// TIA Portal V20 export
FUNCTION_BLOCK "FB_Digital_Output"   // FB3, LAD
{ S7_Optimized_Access := 'TRUE' }
// stored: AutoNumber false, MemoryReserve 100, SetENOAutomatically false
   VAR_INPUT
      DB_In_Emergency_Stop_Release : Bool;
      DB_In_Selected_Voltage_220V : Bool;
      DB_In_Selected_Voltage_127V : Bool;
      DB_Spin_Carousel_Frequency_Inverter_Speed_1 : Bool;
      DB_Spin_Carousel_Frequency_Inverter_Speed_2 : Bool;
      DB_Spin_Carousel_Frequency_Inverter_Speed_3 : Bool;
      DB_Conveyor_Belt_Frequency_Inverter_Speed_1 : Bool;
      DB_Conveyor_Belt_Frequency_Inverter_Speed_2 : Bool;
      DB_Conveyor_Belt_Frequency_Inverter_Speed_3 : Bool;
      DB_Turn_On_Conveyor_Belt_Motor_Spinner_Get_Entrace_Function_Test : Bool;
      DB_Turn_On_Conveyor_Belt_Motor_Rework_Conveyor_Belt_Get_Entrace_Functional_Test : Bool;
      DB_Turn_On_Conveyor_Belt_Motor_Spinner_Get_Exit_Functional_Test : Bool;
      DB_Turn_On_Conveyor_Belt_Motor_Rework_Conveyor_Belt_Get_Exit_Funcional_Test : Bool;
      DB_Open_Air_Pressure : Bool;
      DB_Valve_Advance_Spinner_Get_Entrace_Functional_Test : Bool;
      DB_Valve_Advance_Spinner_Get_Exit_Functional_Test : Bool;
      DB_Signal_Pre_Functional_Test_Production_Line : Bool;
      DB_Digital_Output_14 : Bool;
      DB_Digital_Output_15 : Bool;
      DB_Digital_Output_16 : Bool;
      DB_Digital_Output_17 : Bool;
      DB_Digital_Output_18 : Bool;
      DB_Digital_Output_19 : Bool;
      DB_Digital_Output_20 : Bool;
      DB_Digital_Output_21 : Bool;
      DB_Digital_Output_22 : Bool;
      DB_Digital_Output_23 : Bool;
      DB_Voltage_220V_Selected : Bool;
      DB_Voltage_127V_Selected : Bool;
   END_VAR
   VAR_OUTPUT
      DO_Spin_Carousel_Frequency_Inverter_Speed_1 : Bool;
      DO_Spin_Carousel_Frequency_Inverter_Speed_2 : Bool;
      DO_Spin_Carousel_Frequency_Inverter_Speed_3 : Bool;
      DO_Conveyor_Belt_Frequency_Inverter_Speed_1 : Bool;
      DO_Conveyor_Belt_Frequency_Inverter_Speed_2 : Bool;
      DO_Conveyor_Belt_Frequency_Inverter_Speed_3 : Bool;
      DO_Turn_On_Conveyor_Belt_Motor_Spinner_Get_Entrace_Function_Test : Bool;
      DO_Turn_On_Conveyor_Belt_Motor_Rework_Conveyor_Belt_Get_Entrace_Functional_Test : Bool;
      DO_Turn_On_Conveyor_Belt_Motor_Spinner_Get_Exit_Functional_Test : Bool;
      DO_Turn_On_Conveyor_Belt_Motor_Rework_Conveyor_Belt_Get_Exit_Funcional_Test : Bool;
      DO_Open_Air_Pressure : Bool;
      DO_Valve_Advance_Spinner_Entrace_Functional_Test : Bool;
      DO_Valve_Advance_Spinner_Exit_Functional_Test : Bool;
      DO_Signal_Pre_Functional_Test_Production_Line : Bool;
      DO_Digital_Output_14 : Bool;
      DO_Digital_Output_15 : Bool;
      DO_Digital_Output_16 : Bool;
      DO_Digital_Output_17 : Bool;
      DO_Digital_Output_18 : Bool;
      DO_Digital_Output_19 : Bool;
      DO_Digital_Output_20 : Bool;
      DO_Digital_Output_21 : Bool;
      DO_Digital_Output_22 : Bool;
      DO_Digital_Output_23 : Bool;
      DO_Voltage_220V_Selected : Bool;
      DO_Voltage_127V_Selected : Bool;
   END_VAR
   VAR
      Timer_Delay_Turn_On_220_V { S7_SetPoint := 'True'} : TON_TIME;
      Timer_Delay_Turn_On_127_V { S7_SetPoint := 'True'} : TON_TIME;
   END_VAR
BEGIN

REGION Network 1
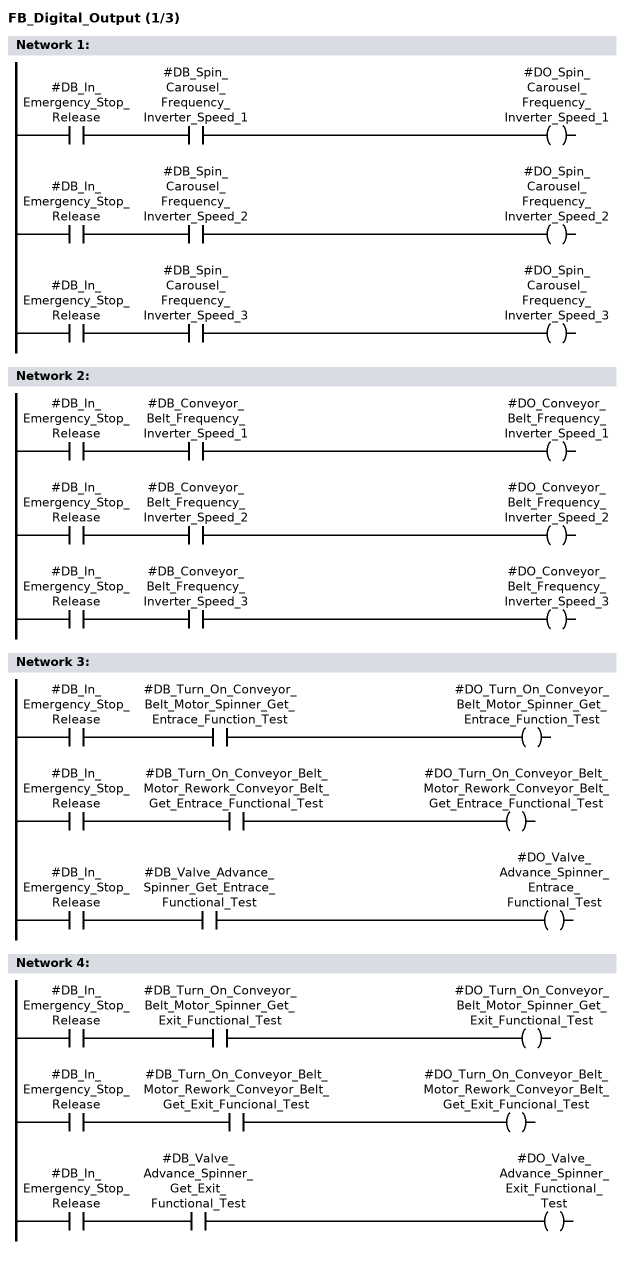
   RUNG wire#powerrail
      Contact( #DB_In_Emergency_Stop_Release )
      Contact( #DB_Spin_Carousel_Frequency_Inverter_Speed_1 )
      Coil( #DO_Spin_Carousel_Frequency_Inverter_Speed_1 )
   END_RUNG
   RUNG wire#powerrail
      Contact( #DB_In_Emergency_Stop_Release )
      Contact( #DB_Spin_Carousel_Frequency_Inverter_Speed_2 )
      Coil( #DO_Spin_Carousel_Frequency_Inverter_Speed_2 )
   END_RUNG
   RUNG wire#powerrail
      Contact( #DB_In_Emergency_Stop_Release )
      Contact( #DB_Spin_Carousel_Frequency_Inverter_Speed_3 )
      Coil( #DO_Spin_Carousel_Frequency_Inverter_Speed_3 )
   END_RUNG
   // the same network as SCL:
   #DO_Spin_Carousel_Frequency_Inverter_Speed_1 := #DB_In_Emergency_Stop_Release AND #DB_Spin_Carousel_Frequency_Inverter_Speed_1;
   #DO_Spin_Carousel_Frequency_Inverter_Speed_2 := #DB_In_Emergency_Stop_Release AND #DB_Spin_Carousel_Frequency_Inverter_Speed_2;
   #DO_Spin_Carousel_Frequency_Inverter_Speed_3 := #DB_In_Emergency_Stop_Release AND #DB_Spin_Carousel_Frequency_Inverter_Speed_3;
END_REGION

REGION Network 2
   RUNG wire#powerrail
      Contact( #DB_In_Emergency_Stop_Release )
      Contact( #DB_Conveyor_Belt_Frequency_Inverter_Speed_1 )
      Coil( #DO_Conveyor_Belt_Frequency_Inverter_Speed_1 )
   END_RUNG
   RUNG wire#powerrail
      Contact( #DB_In_Emergency_Stop_Release )
      Contact( #DB_Conveyor_Belt_Frequency_Inverter_Speed_2 )
      Coil( #DO_Conveyor_Belt_Frequency_Inverter_Speed_2 )
   END_RUNG
   RUNG wire#powerrail
      Contact( #DB_In_Emergency_Stop_Release )
      Contact( #DB_Conveyor_Belt_Frequency_Inverter_Speed_3 )
      Coil( #DO_Conveyor_Belt_Frequency_Inverter_Speed_3 )
   END_RUNG
   // the same network as SCL:
   #DO_Conveyor_Belt_Frequency_Inverter_Speed_1 := #DB_In_Emergency_Stop_Release AND #DB_Conveyor_Belt_Frequency_Inverter_Speed_1;
   #DO_Conveyor_Belt_Frequency_Inverter_Speed_2 := #DB_In_Emergency_Stop_Release AND #DB_Conveyor_Belt_Frequency_Inverter_Speed_2;
   #DO_Conveyor_Belt_Frequency_Inverter_Speed_3 := #DB_In_Emergency_Stop_Release AND #DB_Conveyor_Belt_Frequency_Inverter_Speed_3;
END_REGION

REGION Network 3
   RUNG wire#powerrail
      Contact( #DB_In_Emergency_Stop_Release )
      Contact( #DB_Turn_On_Conveyor_Belt_Motor_Spinner_Get_Entrace_Function_Test )
      Coil( #DO_Turn_On_Conveyor_Belt_Motor_Spinner_Get_Entrace_Function_Test )
   END_RUNG
   RUNG wire#powerrail
      Contact( #DB_In_Emergency_Stop_Release )
      Contact( #DB_Turn_On_Conveyor_Belt_Motor_Rework_Conveyor_Belt_Get_Entrace_Functional_Test )
      Coil( #DO_Turn_On_Conveyor_Belt_Motor_Rework_Conveyor_Belt_Get_Entrace_Functional_Test )
   END_RUNG
   RUNG wire#powerrail
      Contact( #DB_In_Emergency_Stop_Release )
      Contact( #DB_Valve_Advance_Spinner_Get_Entrace_Functional_Test )
      Coil( #DO_Valve_Advance_Spinner_Entrace_Functional_Test )
   END_RUNG
   // the same network as SCL:
   #DO_Turn_On_Conveyor_Belt_Motor_Spinner_Get_Entrace_Function_Test := #DB_In_Emergency_Stop_Release AND #DB_Turn_On_Conveyor_Belt_Motor_Spinner_Get_Entrace_Function_Test;
   #DO_Turn_On_Conveyor_Belt_Motor_Rework_Conveyor_Belt_Get_Entrace_Functional_Test := #DB_In_Emergency_Stop_Release AND #DB_Turn_On_Conveyor_Belt_Motor_Rework_Conveyor_Belt_Get_Entrace_Functional_Test;
   #DO_Valve_Advance_Spinner_Entrace_Functional_Test := #DB_In_Emergency_Stop_Release AND #DB_Valve_Advance_Spinner_Get_Entrace_Functional_Test;
END_REGION

REGION Network 4
   RUNG wire#powerrail
      Contact( #DB_In_Emergency_Stop_Release )
      Contact( #DB_Turn_On_Conveyor_Belt_Motor_Spinner_Get_Exit_Functional_Test )
      Coil( #DO_Turn_On_Conveyor_Belt_Motor_Spinner_Get_Exit_Functional_Test )
   END_RUNG
   RUNG wire#powerrail
      Contact( #DB_In_Emergency_Stop_Release )
      Contact( #DB_Turn_On_Conveyor_Belt_Motor_Rework_Conveyor_Belt_Get_Exit_Funcional_Test )
      Coil( #DO_Turn_On_Conveyor_Belt_Motor_Rework_Conveyor_Belt_Get_Exit_Funcional_Test )
   END_RUNG
   RUNG wire#powerrail
      Contact( #DB_In_Emergency_Stop_Release )
      Contact( #DB_Valve_Advance_Spinner_Get_Exit_Functional_Test )
      Coil( #DO_Valve_Advance_Spinner_Exit_Functional_Test )
   END_RUNG
   // the same network as SCL:
   #DO_Turn_On_Conveyor_Belt_Motor_Spinner_Get_Exit_Functional_Test := #DB_In_Emergency_Stop_Release AND #DB_Turn_On_Conveyor_Belt_Motor_Spinner_Get_Exit_Functional_Test;
   #DO_Turn_On_Conveyor_Belt_Motor_Rework_Conveyor_Belt_Get_Exit_Funcional_Test := #DB_In_Emergency_Stop_Release AND #DB_Turn_On_Conveyor_Belt_Motor_Rework_Conveyor_Belt_Get_Exit_Funcional_Test;
   #DO_Valve_Advance_Spinner_Exit_Functional_Test := #DB_In_Emergency_Stop_Release AND #DB_Valve_Advance_Spinner_Get_Exit_Functional_Test;
END_REGION

REGION Network 5
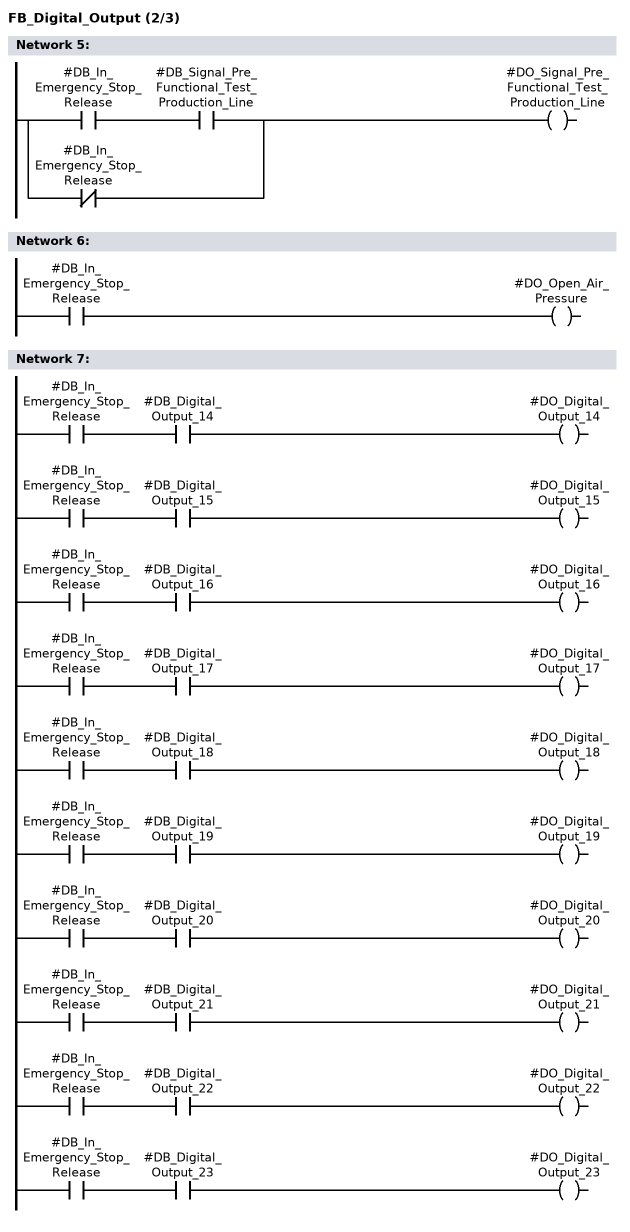
   RUNG wire#powerrail
      Contact( #DB_In_Emergency_Stop_Release )
      Contact( #DB_Signal_Pre_Functional_Test_Production_Line )
      wire#w1
      Coil( #DO_Signal_Pre_Functional_Test_Production_Line )
   END_RUNG
   RUNG wire#powerrail
      I_Contact( #DB_In_Emergency_Stop_Release )
   END_RUNG wire#w1
   // the same network as SCL:
   #DO_Signal_Pre_Functional_Test_Production_Line := (#DB_In_Emergency_Stop_Release AND #DB_Signal_Pre_Functional_Test_Production_Line) OR NOT #DB_In_Emergency_Stop_Release;
END_REGION

REGION Network 6
   RUNG wire#powerrail
      Contact( #DB_In_Emergency_Stop_Release )
      Coil( #DO_Open_Air_Pressure )
   END_RUNG
   // the same network as SCL:
   #DO_Open_Air_Pressure := #DB_In_Emergency_Stop_Release;
END_REGION

REGION Network 7
   RUNG wire#powerrail
      Contact( #DB_In_Emergency_Stop_Release )
      Contact( #DB_Digital_Output_14 )
      Coil( #DO_Digital_Output_14 )
   END_RUNG
   RUNG wire#powerrail
      Contact( #DB_In_Emergency_Stop_Release )
      Contact( #DB_Digital_Output_15 )
      Coil( #DO_Digital_Output_15 )
   END_RUNG
   RUNG wire#powerrail
      Contact( #DB_In_Emergency_Stop_Release )
      Contact( #DB_Digital_Output_16 )
      Coil( #DO_Digital_Output_16 )
   END_RUNG
   RUNG wire#powerrail
      Contact( #DB_In_Emergency_Stop_Release )
      Contact( #DB_Digital_Output_17 )
      Coil( #DO_Digital_Output_17 )
   END_RUNG
   RUNG wire#powerrail
      Contact( #DB_In_Emergency_Stop_Release )
      Contact( #DB_Digital_Output_18 )
      Coil( #DO_Digital_Output_18 )
   END_RUNG
   RUNG wire#powerrail
      Contact( #DB_In_Emergency_Stop_Release )
      Contact( #DB_Digital_Output_19 )
      Coil( #DO_Digital_Output_19 )
   END_RUNG
   RUNG wire#powerrail
      Contact( #DB_In_Emergency_Stop_Release )
      Contact( #DB_Digital_Output_20 )
      Coil( #DO_Digital_Output_20 )
   END_RUNG
   RUNG wire#powerrail
      Contact( #DB_In_Emergency_Stop_Release )
      Contact( #DB_Digital_Output_21 )
      Coil( #DO_Digital_Output_21 )
   END_RUNG
   RUNG wire#powerrail
      Contact( #DB_In_Emergency_Stop_Release )
      Contact( #DB_Digital_Output_22 )
      Coil( #DO_Digital_Output_22 )
   END_RUNG
   RUNG wire#powerrail
      Contact( #DB_In_Emergency_Stop_Release )
      Contact( #DB_Digital_Output_23 )
      Coil( #DO_Digital_Output_23 )
   END_RUNG
   // the same network as SCL:
   #DO_Digital_Output_14 := #DB_In_Emergency_Stop_Release AND #DB_Digital_Output_14;
   #DO_Digital_Output_15 := #DB_In_Emergency_Stop_Release AND #DB_Digital_Output_15;
   #DO_Digital_Output_16 := #DB_In_Emergency_Stop_Release AND #DB_Digital_Output_16;
   #DO_Digital_Output_17 := #DB_In_Emergency_Stop_Release AND #DB_Digital_Output_17;
   #DO_Digital_Output_18 := #DB_In_Emergency_Stop_Release AND #DB_Digital_Output_18;
   #DO_Digital_Output_19 := #DB_In_Emergency_Stop_Release AND #DB_Digital_Output_19;
   #DO_Digital_Output_20 := #DB_In_Emergency_Stop_Release AND #DB_Digital_Output_20;
   #DO_Digital_Output_21 := #DB_In_Emergency_Stop_Release AND #DB_Digital_Output_21;
   #DO_Digital_Output_22 := #DB_In_Emergency_Stop_Release AND #DB_Digital_Output_22;
   #DO_Digital_Output_23 := #DB_In_Emergency_Stop_Release AND #DB_Digital_Output_23;
END_REGION

REGION Network 8
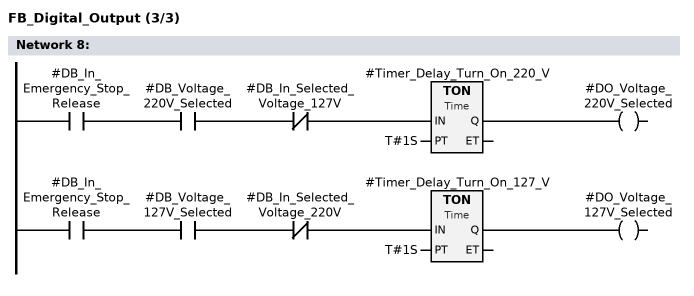
   RUNG wire#powerrail
      Contact( #DB_In_Emergency_Stop_Release )
      Contact( #DB_Voltage_220V_Selected )
      I_Contact( #DB_In_Selected_Voltage_127V )
      { S7_Templates := "time_type := Time" } #Timer_Delay_Turn_On_220_V.TON(pt := T#1S, et =>)
      Coil( #DO_Voltage_220V_Selected )
   END_RUNG
   RUNG wire#powerrail
      Contact( #DB_In_Emergency_Stop_Release )
      Contact( #DB_Voltage_127V_Selected )
      I_Contact( #DB_In_Selected_Voltage_220V )
      { S7_Templates := "time_type := Time" } #Timer_Delay_Turn_On_127_V.TON(pt := T#1S, et =>)
      Coil( #DO_Voltage_127V_Selected )
   END_RUNG
   // the same network as SCL:
   #Timer_Delay_Turn_On_220_V(IN := #DB_In_Emergency_Stop_Release AND #DB_Voltage_220V_Selected AND NOT #DB_In_Selected_Voltage_127V,   // TON
                           PT := T#1S);
   #DO_Voltage_220V_Selected := #Timer_Delay_Turn_On_220_V.Q;
   #Timer_Delay_Turn_On_127_V(IN := #DB_In_Emergency_Stop_Release AND #DB_Voltage_127V_Selected AND NOT #DB_In_Selected_Voltage_220V,   // TON
                           PT := T#1S);
   #DO_Voltage_127V_Selected := #Timer_Delay_Turn_On_127_V.Q;
END_REGION
END_FUNCTION_BLOCK
